{attribute 'qualified_only'}
VAR_GLOBAL
	bAnalog_Outputs AT %Q* : ARRAY[1..2] OF INT;
	Analog_Outputs_Values : ARRAY[1..2] OF REAL;
END_VAR

(* stored: Version 1.1.0.1, ProductVersion 3.1.4024.12
   GVL GVL: Id {c9801d09-e504-47a5-a236-37c9152750c8} *)
